INTERFACE I_VolumeFlowSensor

METHOD Run : BOOL
VAR_INPUT
END_VAR
END_METHOD

PROPERTY VolumeFlow : REAL
GET
END_GET
SET
END_SET
END_PROPERTY

END_INTERFACE

(* stored: Version 1.1.0.1, ProductVersion 3.1.4024.6
   Itf I_VolumeFlowSensor: Id {089227fb-b415-4beb-aaea-251b5d9eb105}
   Method Run: Id {5155f185-d9eb-43d8-88a6-d324b645ae90}
   Property VolumeFlow: Id {2b0f1f59-a34e-49da-a853-6c2b5f240a43}
   Get Get: Id {e649a035-edf1-407f-8052-fd2b698baefe}
   Set Set: Id {86fc4102-6c32-4901-a6a1-8dd00791e016} *)
